TYPE TelemetryAccelerometerConfig :
STRUCT
	///X angle
	x: MeasurementConfig;
	///X angle
	y: MeasurementConfig;
END_STRUCT
END_TYPE

(* stored: Version 1.1.0.1, ProductVersion 3.1.4019.2
   DUT TelemetryAccelerometerConfig: Id {19f428cd-b9ee-404c-afb1-c7739caaf31f} *)
